DATA_BLOCK "Data_block_1"
{ S7_Optimized_Access := 'TRUE' }
VERSION : 0.1
NON_RETAIN
   VAR
      a : Bool;
      a_1 : Bool;
      a_2 : Bool;
   END_VAR
   VAR RETAIN
      a_3 : Bool;
   END_VAR
   VAR
      a_4 { ExternalAccessible := 'False'; ExternalVisible := 'False'; ExternalWritable := 'False'} : Bool;
      a_5 : Bool;
      a_6 { ExternalWritable := 'False'} : Bool;
      a_7 : Array[0..10000] of Int;
      a_8 { ExternalVisible := 'False'; ExternalWritable := 'False'} : Bool;
   END_VAR
   VAR RETAIN
      a_9 : Bool;
   END_VAR
   VAR
      a_10 : Bool;
   END_VAR


BEGIN

END_DATA_BLOCK

